// TIA Portal V20 export
ORGANIZATION_BLOCK "Startup"   // OB100, LAD, Startup
TITLE = "Complete Restart"
// stored: AutoNumber false, IsIECCheckEnabled true, SetENOAutomatically true
   VAR_INPUT
      LostRetentive : Bool;   // True if retentive data are lost
      LostRTC : Bool;   // True if date and time are lost
   END_VAR
   VAR_TEMP
      tempError : Bool;
      tempStatus : Word;
      tempDiagnostics : "LAF_typeDiagnosticsSimple";
   END_VAR
BEGIN

REGION Network 1: Set first cycle bit
   // Set the first cycle signal
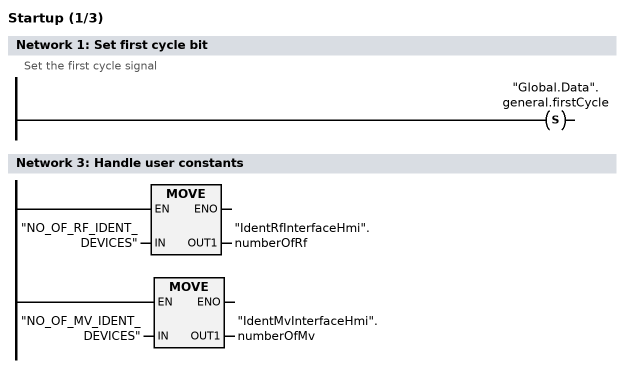
   RUNG wire#powerrail
      S_Coil( "Global.Data".general.firstCycle )
   END_RUNG
   // the same network as SCL:
   "Global.Data".general.firstCycle := TRUE;
END_REGION

REGION Network 2: Enable global power
   // Set global power to true by default. This can be adjusted depending on the user requirement for a specific machine.
END_REGION

REGION Network 3: Handle user constants
   RUNG wire#powerrail
      Move(in := "NO_OF_RF_IDENT_DEVICES", out1 => "IdentRfInterfaceHmi".numberOfRf)
   END_RUNG
   RUNG wire#powerrail
      Move(in := "NO_OF_MV_IDENT_DEVICES", out1 => "IdentMvInterfaceHmi".numberOfMv)
   END_RUNG
   // the same network as SCL:
   "IdentRfInterfaceHmi".numberOfRf := "NO_OF_RF_IDENT_DEVICES";
   "IdentMvInterfaceHmi".numberOfMv := "NO_OF_MV_IDENT_DEVICES";
END_REGION

REGION Network 4: Set drive objects for drive diagnostic
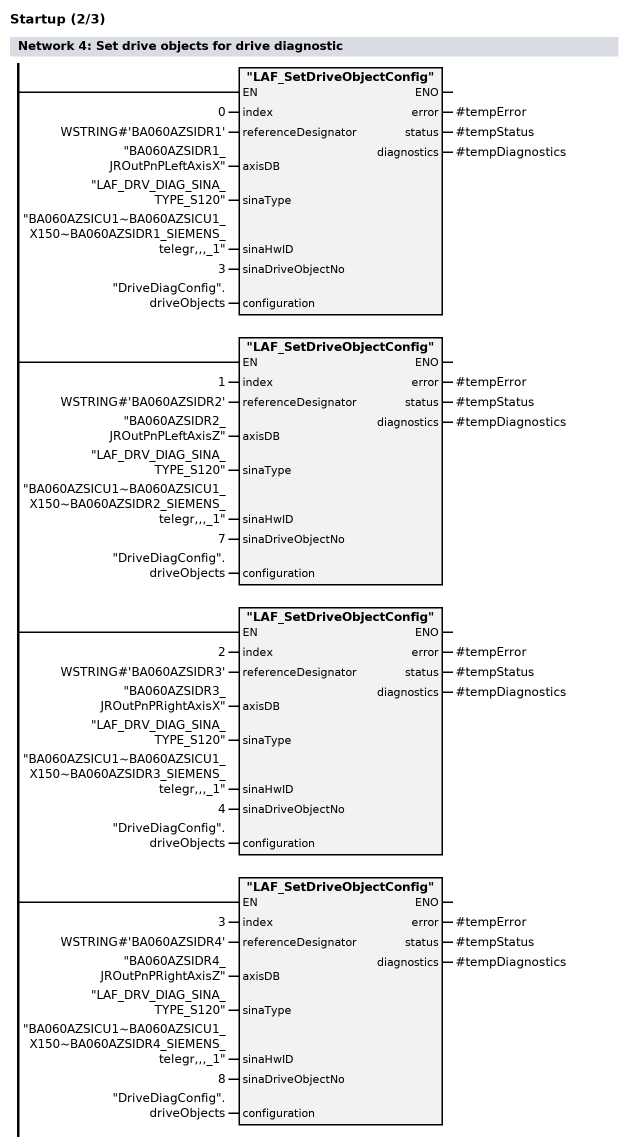
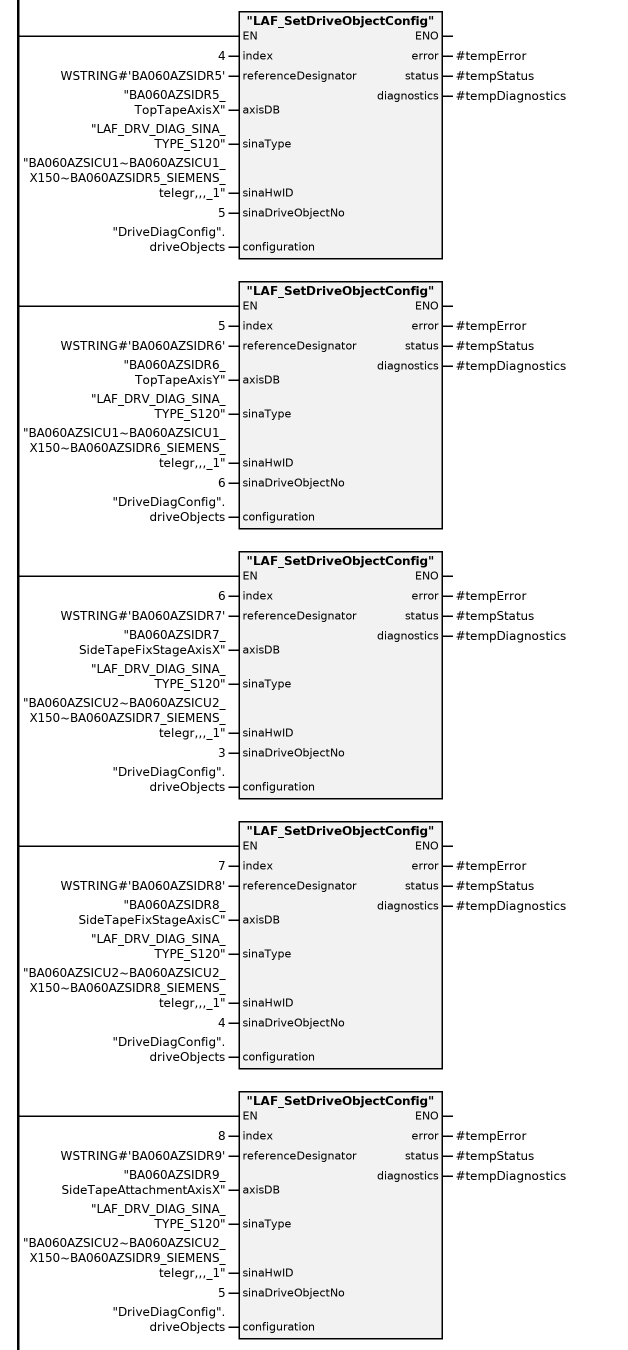
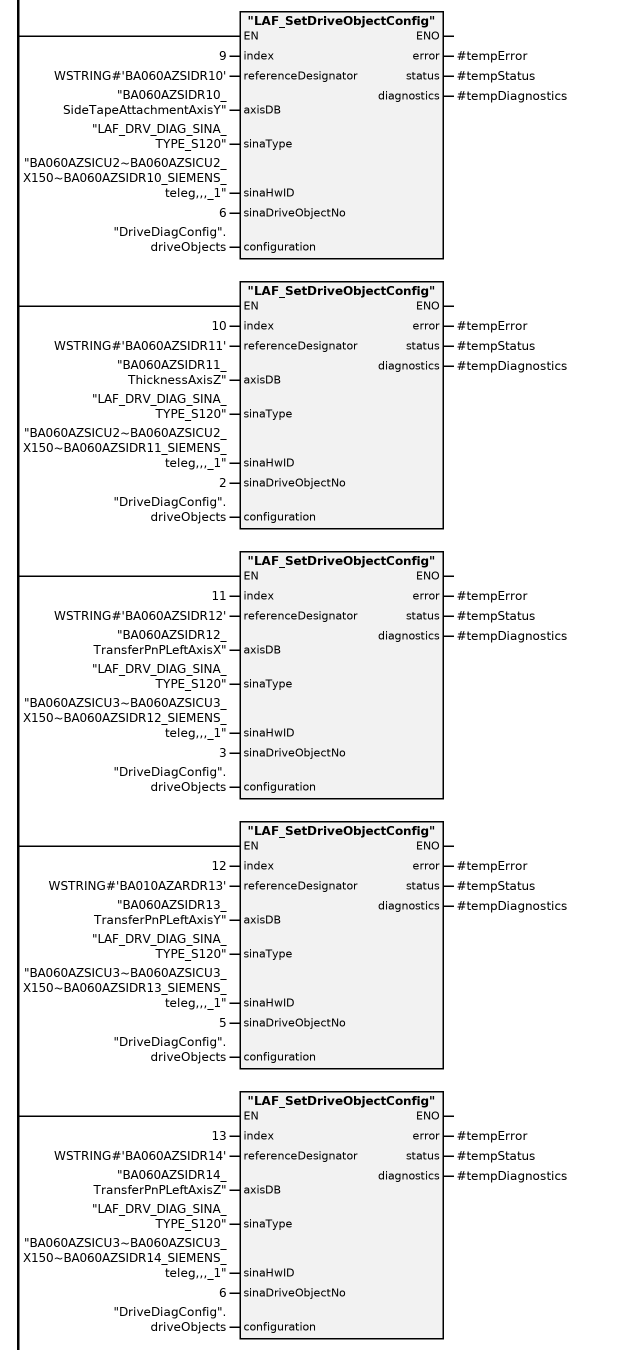
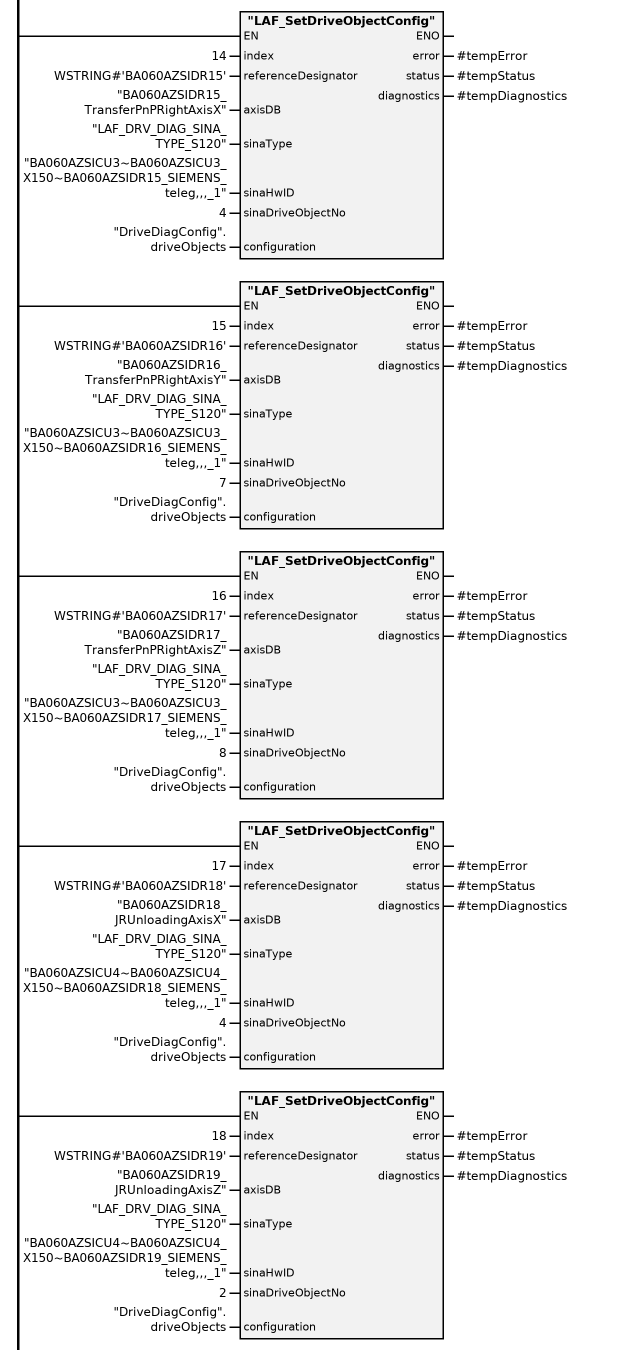
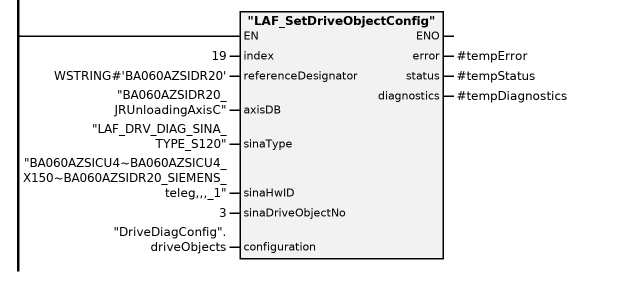
   RUNG wire#powerrail
      "LAF_SetDriveObjectConfig"(index := 0, referenceDesignator := WSTRING#'BA060AZSIDR1', axisDB := "BA060AZSIDR1_JROutPnPLeftAxisX", sinaType := "LAF_DRV_DIAG_SINA_TYPE_S120", sinaHwID := "BA060AZSICU1~BA060AZSICU1_X150~BA060AZSIDR1_SIEMENS_telegr,,,_1", sinaDriveObjectNo := 3, configuration := "DriveDiagConfig".driveObjects, error => #tempError, status => #tempStatus, diagnostics => #tempDiagnostics)
   END_RUNG
   RUNG wire#powerrail
      "LAF_SetDriveObjectConfig"(index := 1, referenceDesignator := WSTRING#'BA060AZSIDR2', axisDB := "BA060AZSIDR2_JROutPnPLeftAxisZ", sinaType := "LAF_DRV_DIAG_SINA_TYPE_S120", sinaHwID := "BA060AZSICU1~BA060AZSICU1_X150~BA060AZSIDR2_SIEMENS_telegr,,,_1", sinaDriveObjectNo := 7, configuration := "DriveDiagConfig".driveObjects, error => #tempError, status => #tempStatus, diagnostics => #tempDiagnostics)
   END_RUNG
   RUNG wire#powerrail
      "LAF_SetDriveObjectConfig"(index := 2, referenceDesignator := WSTRING#'BA060AZSIDR3', axisDB := "BA060AZSIDR3_JROutPnPRightAxisX", sinaType := "LAF_DRV_DIAG_SINA_TYPE_S120", sinaHwID := "BA060AZSICU1~BA060AZSICU1_X150~BA060AZSIDR3_SIEMENS_telegr,,,_1", sinaDriveObjectNo := 4, configuration := "DriveDiagConfig".driveObjects, error => #tempError, status => #tempStatus, diagnostics => #tempDiagnostics)
   END_RUNG
   RUNG wire#powerrail
      "LAF_SetDriveObjectConfig"(index := 3, referenceDesignator := WSTRING#'BA060AZSIDR4', axisDB := "BA060AZSIDR4_JROutPnPRightAxisZ", sinaType := "LAF_DRV_DIAG_SINA_TYPE_S120", sinaHwID := "BA060AZSICU1~BA060AZSICU1_X150~BA060AZSIDR4_SIEMENS_telegr,,,_1", sinaDriveObjectNo := 8, configuration := "DriveDiagConfig".driveObjects, error => #tempError, status => #tempStatus, diagnostics => #tempDiagnostics)
   END_RUNG
   RUNG wire#powerrail
      "LAF_SetDriveObjectConfig"(index := 4, referenceDesignator := WSTRING#'BA060AZSIDR5', axisDB := "BA060AZSIDR5_TopTapeAxisX", sinaType := "LAF_DRV_DIAG_SINA_TYPE_S120", sinaHwID := "BA060AZSICU1~BA060AZSICU1_X150~BA060AZSIDR5_SIEMENS_telegr,,,_1", sinaDriveObjectNo := 5, configuration := "DriveDiagConfig".driveObjects, error => #tempError, status => #tempStatus, diagnostics => #tempDiagnostics)
   END_RUNG
   RUNG wire#powerrail
      "LAF_SetDriveObjectConfig"(index := 5, referenceDesignator := WSTRING#'BA060AZSIDR6', axisDB := "BA060AZSIDR6_TopTapeAxisY", sinaType := "LAF_DRV_DIAG_SINA_TYPE_S120", sinaHwID := "BA060AZSICU1~BA060AZSICU1_X150~BA060AZSIDR6_SIEMENS_telegr,,,_1", sinaDriveObjectNo := 6, configuration := "DriveDiagConfig".driveObjects, error => #tempError, status => #tempStatus, diagnostics => #tempDiagnostics)
   END_RUNG
   RUNG wire#powerrail
      "LAF_SetDriveObjectConfig"(index := 6, referenceDesignator := WSTRING#'BA060AZSIDR7', axisDB := "BA060AZSIDR7_SideTapeFixStageAxisX", sinaType := "LAF_DRV_DIAG_SINA_TYPE_S120", sinaHwID := "BA060AZSICU2~BA060AZSICU2_X150~BA060AZSIDR7_SIEMENS_telegr,,,_1", sinaDriveObjectNo := 3, configuration := "DriveDiagConfig".driveObjects, error => #tempError, status => #tempStatus, diagnostics => #tempDiagnostics)
   END_RUNG
   RUNG wire#powerrail
      "LAF_SetDriveObjectConfig"(index := 7, referenceDesignator := WSTRING#'BA060AZSIDR8', axisDB := "BA060AZSIDR8_SideTapeFixStageAxisC", sinaType := "LAF_DRV_DIAG_SINA_TYPE_S120", sinaHwID := "BA060AZSICU2~BA060AZSICU2_X150~BA060AZSIDR8_SIEMENS_telegr,,,_1", sinaDriveObjectNo := 4, configuration := "DriveDiagConfig".driveObjects, error => #tempError, status => #tempStatus, diagnostics => #tempDiagnostics)
   END_RUNG
   RUNG wire#powerrail
      "LAF_SetDriveObjectConfig"(index := 8, referenceDesignator := WSTRING#'BA060AZSIDR9', axisDB := "BA060AZSIDR9_SideTapeAttachmentAxisX", sinaType := "LAF_DRV_DIAG_SINA_TYPE_S120", sinaHwID := "BA060AZSICU2~BA060AZSICU2_X150~BA060AZSIDR9_SIEMENS_telegr,,,_1", sinaDriveObjectNo := 5, configuration := "DriveDiagConfig".driveObjects, error => #tempError, status => #tempStatus, diagnostics => #tempDiagnostics)
   END_RUNG
   RUNG wire#powerrail
      "LAF_SetDriveObjectConfig"(index := 9, referenceDesignator := WSTRING#'BA060AZSIDR10', axisDB := "BA060AZSIDR10_SideTapeAttachmentAxisY", sinaType := "LAF_DRV_DIAG_SINA_TYPE_S120", sinaHwID := "BA060AZSICU2~BA060AZSICU2_X150~BA060AZSIDR10_SIEMENS_teleg,,,_1", sinaDriveObjectNo := 6, configuration := "DriveDiagConfig".driveObjects, error => #tempError, status => #tempStatus, diagnostics => #tempDiagnostics)
   END_RUNG
   RUNG wire#powerrail
      "LAF_SetDriveObjectConfig"(index := 10, referenceDesignator := WSTRING#'BA060AZSIDR11', axisDB := "BA060AZSIDR11_ThicknessAxisZ", sinaType := "LAF_DRV_DIAG_SINA_TYPE_S120", sinaHwID := "BA060AZSICU2~BA060AZSICU2_X150~BA060AZSIDR11_SIEMENS_teleg,,,_1", sinaDriveObjectNo := 2, configuration := "DriveDiagConfig".driveObjects, error => #tempError, status => #tempStatus, diagnostics => #tempDiagnostics)
   END_RUNG
   RUNG wire#powerrail
      "LAF_SetDriveObjectConfig"(index := 11, referenceDesignator := WSTRING#'BA060AZSIDR12', axisDB := "BA060AZSIDR12_TransferPnPLeftAxisX", sinaType := "LAF_DRV_DIAG_SINA_TYPE_S120", sinaHwID := "BA060AZSICU3~BA060AZSICU3_X150~BA060AZSIDR12_SIEMENS_teleg,,,_1", sinaDriveObjectNo := 3, configuration := "DriveDiagConfig".driveObjects, error => #tempError, status => #tempStatus, diagnostics => #tempDiagnostics)
   END_RUNG
   RUNG wire#powerrail
      "LAF_SetDriveObjectConfig"(index := 12, referenceDesignator := WSTRING#'BA010AZARDR13', axisDB := "BA060AZSIDR13_TransferPnPLeftAxisY", sinaType := "LAF_DRV_DIAG_SINA_TYPE_S120", sinaHwID := "BA060AZSICU3~BA060AZSICU3_X150~BA060AZSIDR13_SIEMENS_teleg,,,_1", sinaDriveObjectNo := 5, configuration := "DriveDiagConfig".driveObjects, error => #tempError, status => #tempStatus, diagnostics => #tempDiagnostics)
   END_RUNG
   RUNG wire#powerrail
      "LAF_SetDriveObjectConfig"(index := 13, referenceDesignator := WSTRING#'BA060AZSIDR14', axisDB := "BA060AZSIDR14_TransferPnPLeftAxisZ", sinaType := "LAF_DRV_DIAG_SINA_TYPE_S120", sinaHwID := "BA060AZSICU3~BA060AZSICU3_X150~BA060AZSIDR14_SIEMENS_teleg,,,_1", sinaDriveObjectNo := 6, configuration := "DriveDiagConfig".driveObjects, error => #tempError, status => #tempStatus, diagnostics => #tempDiagnostics)
   END_RUNG
   RUNG wire#powerrail
      "LAF_SetDriveObjectConfig"(index := 14, referenceDesignator := WSTRING#'BA060AZSIDR15', axisDB := "BA060AZSIDR15_TransferPnPRightAxisX", sinaType := "LAF_DRV_DIAG_SINA_TYPE_S120", sinaHwID := "BA060AZSICU3~BA060AZSICU3_X150~BA060AZSIDR15_SIEMENS_teleg,,,_1", sinaDriveObjectNo := 4, configuration := "DriveDiagConfig".driveObjects, error => #tempError, status => #tempStatus, diagnostics => #tempDiagnostics)
   END_RUNG
   RUNG wire#powerrail
      "LAF_SetDriveObjectConfig"(index := 15, referenceDesignator := WSTRING#'BA060AZSIDR16', axisDB := "BA060AZSIDR16_TransferPnPRightAxisY", sinaType := "LAF_DRV_DIAG_SINA_TYPE_S120", sinaHwID := "BA060AZSICU3~BA060AZSICU3_X150~BA060AZSIDR16_SIEMENS_teleg,,,_1", sinaDriveObjectNo := 7, configuration := "DriveDiagConfig".driveObjects, error => #tempError, status => #tempStatus, diagnostics => #tempDiagnostics)
   END_RUNG
   RUNG wire#powerrail
      "LAF_SetDriveObjectConfig"(index := 16, referenceDesignator := WSTRING#'BA060AZSIDR17', axisDB := "BA060AZSIDR17_TransferPnPRightAxisZ", sinaType := "LAF_DRV_DIAG_SINA_TYPE_S120", sinaHwID := "BA060AZSICU3~BA060AZSICU3_X150~BA060AZSIDR17_SIEMENS_teleg,,,_1", sinaDriveObjectNo := 8, configuration := "DriveDiagConfig".driveObjects, error => #tempError, status => #tempStatus, diagnostics => #tempDiagnostics)
   END_RUNG
   RUNG wire#powerrail
      "LAF_SetDriveObjectConfig"(index := 17, referenceDesignator := WSTRING#'BA060AZSIDR18', axisDB := "BA060AZSIDR18_JRUnloadingAxisX", sinaType := "LAF_DRV_DIAG_SINA_TYPE_S120", sinaHwID := "BA060AZSICU4~BA060AZSICU4_X150~BA060AZSIDR18_SIEMENS_teleg,,,_1", sinaDriveObjectNo := 4, configuration := "DriveDiagConfig".driveObjects, error => #tempError, status => #tempStatus, diagnostics => #tempDiagnostics)
   END_RUNG
   RUNG wire#powerrail
      "LAF_SetDriveObjectConfig"(index := 18, referenceDesignator := WSTRING#'BA060AZSIDR19', axisDB := "BA060AZSIDR19_JRUnloadingAxisZ", sinaType := "LAF_DRV_DIAG_SINA_TYPE_S120", sinaHwID := "BA060AZSICU4~BA060AZSICU4_X150~BA060AZSIDR19_SIEMENS_teleg,,,_1", sinaDriveObjectNo := 2, configuration := "DriveDiagConfig".driveObjects, error => #tempError, status => #tempStatus, diagnostics => #tempDiagnostics)
   END_RUNG
   RUNG wire#powerrail
      "LAF_SetDriveObjectConfig"(index := 19, referenceDesignator := WSTRING#'BA060AZSIDR20', axisDB := "BA060AZSIDR20_JRUnloadingAxisC", sinaType := "LAF_DRV_DIAG_SINA_TYPE_S120", sinaHwID := "BA060AZSICU4~BA060AZSICU4_X150~BA060AZSIDR20_SIEMENS_teleg,,,_1", sinaDriveObjectNo := 3, configuration := "DriveDiagConfig".driveObjects, error => #tempError, status => #tempStatus, diagnostics => #tempDiagnostics)
   END_RUNG
   // the same network as SCL:
   "LAF_SetDriveObjectConfig"(index := 0,
                           referenceDesignator := WSTRING#'BA060AZSIDR1',
                           axisDB := "BA060AZSIDR1_JROutPnPLeftAxisX",
                           sinaType := "LAF_DRV_DIAG_SINA_TYPE_S120",
                           sinaHwID := "BA060AZSICU1~BA060AZSICU1_X150~BA060AZSIDR1_SIEMENS_telegr,,,_1",
                           sinaDriveObjectNo := 3,
                           configuration := "DriveDiagConfig".driveObjects,
                           error => #tempError,
                           status => #tempStatus,
                           diagnostics => #tempDiagnostics);
   "LAF_SetDriveObjectConfig"(index := 1,
                           referenceDesignator := WSTRING#'BA060AZSIDR2',
                           axisDB := "BA060AZSIDR2_JROutPnPLeftAxisZ",
                           sinaType := "LAF_DRV_DIAG_SINA_TYPE_S120",
                           sinaHwID := "BA060AZSICU1~BA060AZSICU1_X150~BA060AZSIDR2_SIEMENS_telegr,,,_1",
                           sinaDriveObjectNo := 7,
                           configuration := "DriveDiagConfig".driveObjects,
                           error => #tempError,
                           status => #tempStatus,
                           diagnostics => #tempDiagnostics);
   "LAF_SetDriveObjectConfig"(index := 2,
                           referenceDesignator := WSTRING#'BA060AZSIDR3',
                           axisDB := "BA060AZSIDR3_JROutPnPRightAxisX",
                           sinaType := "LAF_DRV_DIAG_SINA_TYPE_S120",
                           sinaHwID := "BA060AZSICU1~BA060AZSICU1_X150~BA060AZSIDR3_SIEMENS_telegr,,,_1",
                           sinaDriveObjectNo := 4,
                           configuration := "DriveDiagConfig".driveObjects,
                           error => #tempError,
                           status => #tempStatus,
                           diagnostics => #tempDiagnostics);
   "LAF_SetDriveObjectConfig"(index := 3,
                           referenceDesignator := WSTRING#'BA060AZSIDR4',
                           axisDB := "BA060AZSIDR4_JROutPnPRightAxisZ",
                           sinaType := "LAF_DRV_DIAG_SINA_TYPE_S120",
                           sinaHwID := "BA060AZSICU1~BA060AZSICU1_X150~BA060AZSIDR4_SIEMENS_telegr,,,_1",
                           sinaDriveObjectNo := 8,
                           configuration := "DriveDiagConfig".driveObjects,
                           error => #tempError,
                           status => #tempStatus,
                           diagnostics => #tempDiagnostics);
   "LAF_SetDriveObjectConfig"(index := 4,
                           referenceDesignator := WSTRING#'BA060AZSIDR5',
                           axisDB := "BA060AZSIDR5_TopTapeAxisX",
                           sinaType := "LAF_DRV_DIAG_SINA_TYPE_S120",
                           sinaHwID := "BA060AZSICU1~BA060AZSICU1_X150~BA060AZSIDR5_SIEMENS_telegr,,,_1",
                           sinaDriveObjectNo := 5,
                           configuration := "DriveDiagConfig".driveObjects,
                           error => #tempError,
                           status => #tempStatus,
                           diagnostics => #tempDiagnostics);
   "LAF_SetDriveObjectConfig"(index := 5,
                           referenceDesignator := WSTRING#'BA060AZSIDR6',
                           axisDB := "BA060AZSIDR6_TopTapeAxisY",
                           sinaType := "LAF_DRV_DIAG_SINA_TYPE_S120",
                           sinaHwID := "BA060AZSICU1~BA060AZSICU1_X150~BA060AZSIDR6_SIEMENS_telegr,,,_1",
                           sinaDriveObjectNo := 6,
                           configuration := "DriveDiagConfig".driveObjects,
                           error => #tempError,
                           status => #tempStatus,
                           diagnostics => #tempDiagnostics);
   "LAF_SetDriveObjectConfig"(index := 6,
                           referenceDesignator := WSTRING#'BA060AZSIDR7',
                           axisDB := "BA060AZSIDR7_SideTapeFixStageAxisX",
                           sinaType := "LAF_DRV_DIAG_SINA_TYPE_S120",
                           sinaHwID := "BA060AZSICU2~BA060AZSICU2_X150~BA060AZSIDR7_SIEMENS_telegr,,,_1",
                           sinaDriveObjectNo := 3,
                           configuration := "DriveDiagConfig".driveObjects,
                           error => #tempError,
                           status => #tempStatus,
                           diagnostics => #tempDiagnostics);
   "LAF_SetDriveObjectConfig"(index := 7,
                           referenceDesignator := WSTRING#'BA060AZSIDR8',
                           axisDB := "BA060AZSIDR8_SideTapeFixStageAxisC",
                           sinaType := "LAF_DRV_DIAG_SINA_TYPE_S120",
                           sinaHwID := "BA060AZSICU2~BA060AZSICU2_X150~BA060AZSIDR8_SIEMENS_telegr,,,_1",
                           sinaDriveObjectNo := 4,
                           configuration := "DriveDiagConfig".driveObjects,
                           error => #tempError,
                           status => #tempStatus,
                           diagnostics => #tempDiagnostics);
   "LAF_SetDriveObjectConfig"(index := 8,
                           referenceDesignator := WSTRING#'BA060AZSIDR9',
                           axisDB := "BA060AZSIDR9_SideTapeAttachmentAxisX",
                           sinaType := "LAF_DRV_DIAG_SINA_TYPE_S120",
                           sinaHwID := "BA060AZSICU2~BA060AZSICU2_X150~BA060AZSIDR9_SIEMENS_telegr,,,_1",
                           sinaDriveObjectNo := 5,
                           configuration := "DriveDiagConfig".driveObjects,
                           error => #tempError,
                           status => #tempStatus,
                           diagnostics => #tempDiagnostics);
   "LAF_SetDriveObjectConfig"(index := 9,
                           referenceDesignator := WSTRING#'BA060AZSIDR10',
                           axisDB := "BA060AZSIDR10_SideTapeAttachmentAxisY",
                           sinaType := "LAF_DRV_DIAG_SINA_TYPE_S120",
                           sinaHwID := "BA060AZSICU2~BA060AZSICU2_X150~BA060AZSIDR10_SIEMENS_teleg,,,_1",
                           sinaDriveObjectNo := 6,
                           configuration := "DriveDiagConfig".driveObjects,
                           error => #tempError,
                           status => #tempStatus,
                           diagnostics => #tempDiagnostics);
   "LAF_SetDriveObjectConfig"(index := 10,
                           referenceDesignator := WSTRING#'BA060AZSIDR11',
                           axisDB := "BA060AZSIDR11_ThicknessAxisZ",
                           sinaType := "LAF_DRV_DIAG_SINA_TYPE_S120",
                           sinaHwID := "BA060AZSICU2~BA060AZSICU2_X150~BA060AZSIDR11_SIEMENS_teleg,,,_1",
                           sinaDriveObjectNo := 2,
                           configuration := "DriveDiagConfig".driveObjects,
                           error => #tempError,
                           status => #tempStatus,
                           diagnostics => #tempDiagnostics);
   "LAF_SetDriveObjectConfig"(index := 11,
                           referenceDesignator := WSTRING#'BA060AZSIDR12',
                           axisDB := "BA060AZSIDR12_TransferPnPLeftAxisX",
                           sinaType := "LAF_DRV_DIAG_SINA_TYPE_S120",
                           sinaHwID := "BA060AZSICU3~BA060AZSICU3_X150~BA060AZSIDR12_SIEMENS_teleg,,,_1",
                           sinaDriveObjectNo := 3,
                           configuration := "DriveDiagConfig".driveObjects,
                           error => #tempError,
                           status => #tempStatus,
                           diagnostics => #tempDiagnostics);
   "LAF_SetDriveObjectConfig"(index := 12,
                           referenceDesignator := WSTRING#'BA010AZARDR13',
                           axisDB := "BA060AZSIDR13_TransferPnPLeftAxisY",
                           sinaType := "LAF_DRV_DIAG_SINA_TYPE_S120",
                           sinaHwID := "BA060AZSICU3~BA060AZSICU3_X150~BA060AZSIDR13_SIEMENS_teleg,,,_1",
                           sinaDriveObjectNo := 5,
                           configuration := "DriveDiagConfig".driveObjects,
                           error => #tempError,
                           status => #tempStatus,
                           diagnostics => #tempDiagnostics);
   "LAF_SetDriveObjectConfig"(index := 13,
                           referenceDesignator := WSTRING#'BA060AZSIDR14',
                           axisDB := "BA060AZSIDR14_TransferPnPLeftAxisZ",
                           sinaType := "LAF_DRV_DIAG_SINA_TYPE_S120",
                           sinaHwID := "BA060AZSICU3~BA060AZSICU3_X150~BA060AZSIDR14_SIEMENS_teleg,,,_1",
                           sinaDriveObjectNo := 6,
                           configuration := "DriveDiagConfig".driveObjects,
                           error => #tempError,
                           status => #tempStatus,
                           diagnostics => #tempDiagnostics);
   "LAF_SetDriveObjectConfig"(index := 14,
                           referenceDesignator := WSTRING#'BA060AZSIDR15',
                           axisDB := "BA060AZSIDR15_TransferPnPRightAxisX",
                           sinaType := "LAF_DRV_DIAG_SINA_TYPE_S120",
                           sinaHwID := "BA060AZSICU3~BA060AZSICU3_X150~BA060AZSIDR15_SIEMENS_teleg,,,_1",
                           sinaDriveObjectNo := 4,
                           configuration := "DriveDiagConfig".driveObjects,
                           error => #tempError,
                           status => #tempStatus,
                           diagnostics => #tempDiagnostics);
   "LAF_SetDriveObjectConfig"(index := 15,
                           referenceDesignator := WSTRING#'BA060AZSIDR16',
                           axisDB := "BA060AZSIDR16_TransferPnPRightAxisY",
                           sinaType := "LAF_DRV_DIAG_SINA_TYPE_S120",
                           sinaHwID := "BA060AZSICU3~BA060AZSICU3_X150~BA060AZSIDR16_SIEMENS_teleg,,,_1",
                           sinaDriveObjectNo := 7,
                           configuration := "DriveDiagConfig".driveObjects,
                           error => #tempError,
                           status => #tempStatus,
                           diagnostics => #tempDiagnostics);
   "LAF_SetDriveObjectConfig"(index := 16,
                           referenceDesignator := WSTRING#'BA060AZSIDR17',
                           axisDB := "BA060AZSIDR17_TransferPnPRightAxisZ",
                           sinaType := "LAF_DRV_DIAG_SINA_TYPE_S120",
                           sinaHwID := "BA060AZSICU3~BA060AZSICU3_X150~BA060AZSIDR17_SIEMENS_teleg,,,_1",
                           sinaDriveObjectNo := 8,
                           configuration := "DriveDiagConfig".driveObjects,
                           error => #tempError,
                           status => #tempStatus,
                           diagnostics => #tempDiagnostics);
   "LAF_SetDriveObjectConfig"(index := 17,
                           referenceDesignator := WSTRING#'BA060AZSIDR18',
                           axisDB := "BA060AZSIDR18_JRUnloadingAxisX",
                           sinaType := "LAF_DRV_DIAG_SINA_TYPE_S120",
                           sinaHwID := "BA060AZSICU4~BA060AZSICU4_X150~BA060AZSIDR18_SIEMENS_teleg,,,_1",
                           sinaDriveObjectNo := 4,
                           configuration := "DriveDiagConfig".driveObjects,
                           error => #tempError,
                           status => #tempStatus,
                           diagnostics => #tempDiagnostics);
   "LAF_SetDriveObjectConfig"(index := 18,
                           referenceDesignator := WSTRING#'BA060AZSIDR19',
                           axisDB := "BA060AZSIDR19_JRUnloadingAxisZ",
                           sinaType := "LAF_DRV_DIAG_SINA_TYPE_S120",
                           sinaHwID := "BA060AZSICU4~BA060AZSICU4_X150~BA060AZSIDR19_SIEMENS_teleg,,,_1",
                           sinaDriveObjectNo := 2,
                           configuration := "DriveDiagConfig".driveObjects,
                           error => #tempError,
                           status => #tempStatus,
                           diagnostics => #tempDiagnostics);
   "LAF_SetDriveObjectConfig"(index := 19,
                           referenceDesignator := WSTRING#'BA060AZSIDR20',
                           axisDB := "BA060AZSIDR20_JRUnloadingAxisC",
                           sinaType := "LAF_DRV_DIAG_SINA_TYPE_S120",
                           sinaHwID := "BA060AZSICU4~BA060AZSICU4_X150~BA060AZSIDR20_SIEMENS_teleg,,,_1",
                           sinaDriveObjectNo := 3,
                           configuration := "DriveDiagConfig".driveObjects,
                           error => #tempError,
                           status => #tempStatus,
                           diagnostics => #tempDiagnostics);
END_REGION

REGION Network 5: Manual Operation Line
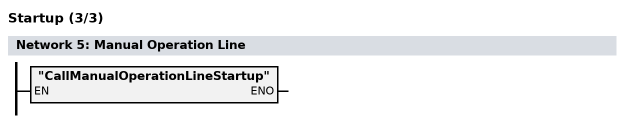
   RUNG wire#powerrail
      "CallManualOperationLineStartup"()
   END_RUNG
   // the same network as SCL:
   "CallManualOperationLineStartup"();
END_REGION

REGION Network 6 (SCL): Configuration Set Position
   //DR01
   "Unit1.Em2.HmiInterface".cmJROutPnPLeftAxisX.configuration.setPositions := "AxisDataBackUp_DB".DR1."configuration.setPositions";
   //Unit1.Em2.HmiInterface.cm.softcam.jrOutPnPLeftAxisX := "AxisDataBackUp_DB".DR1.softcam;


   //DR02
   "Unit1.Em2.HmiInterface".cmJROutPnPLeftAxisZ.configuration.setPositions := "AxisDataBackUp_DB".DR2."configuration.setPositions";
   //Unit1.Em2.HmiInterface.cm.softcam.jrOutPnPLeftAxisZ := "AxisDataBackUp_DB".DR2.softcam;


   //DR03
   "Unit1.Em2.HmiInterface".cmJROutPnPRightAxisX.configuration.setPositions := "AxisDataBackUp_DB".DR3."configuration.setPositions";
   //Unit1.Em2.HmiInterface.cm.softcam.jrOutPnPRightAxisX := "AxisDataBackUp_DB".DR3.softcam;


   //DR04
   "Unit1.Em2.HmiInterface".cmJROutPnPRightAxisZ.configuration.setPositions := "AxisDataBackUp_DB".DR4."configuration.setPositions";
   //Unit1.Em2.HmiInterface.cm.softcam.jrOutPnPRightAxisZ := "AxisDataBackUp_DB".DR4.softcam;


   //DR05
   "Unit1.Em3.HmiInterface".cmTopTapeAxisX.configuration.setPositions := "AxisDataBackUp_DB".DR5."configuration.setPositions";
   //Unit1.Em3.HmiInterface.cm.softcam.topTapeAxisX := "AxisDataBackUp_DB".DR5.softcam;


   //DR06
   "Unit1.Em3.HmiInterface".cmTopTapeAxisY.configuration.setPositions := "AxisDataBackUp_DB".DR6."configuration.setPositions";
   //Unit1.Em3.HmiInterface.cm.softcam.topTapeAxisY := "AxisDataBackUp_DB".DR6.softcam;


   //DR07
   "Unit1.Em4.HmiInterface".cmSideTapeFixStageAxisX.configuration.setPositions := "AxisDataBackUp_DB".DR7."configuration.setPositions";
   //Unit1.Em4.HmiInterface.cm.softcam.sideTapeFixStageAxisX := "AxisDataBackUp_DB".DR7.softcam;


   //DR08
   "Unit1.Em4.HmiInterface".cmSideTapeFixStageAxisC.configuration.setPositions := "AxisDataBackUp_DB".DR8."configuration.setPositions";
   //Unit1.Em4.HmiInterface.cm.softcam.sideTapeFixStageAxisC := "AxisDataBackUp_DB".DR8.softcam;


   //DR09
   "Unit1.Em4.HmiInterface".cmSideTapeAttachmentAxisX.configuration.setPositions := "AxisDataBackUp_DB".DR9."configuration.setPositions";
   //Unit1.Em4.HmiInterface.cm.softcam.sideTapeAttachmentAxisX := "AxisDataBackUp_DB".DR9.softcam;


   //DR10
   "Unit1.Em4.HmiInterface".cmSideTapeAttachmentAxisY.configuration.setPositions := "AxisDataBackUp_DB".DR10."configuration.setPositions";
   //Unit1.Em4.HmiInterface.cm.softcam.sideTapeAttachmentAxisY := "AxisDataBackUp_DB".DR10.softcam;


   //DR11
   "Unit1.Em8.HmiInterface".cmThicknessAxisZ.configuration.setPositions := "AxisDataBackUp_DB".DR11."configuration.setPositions";
   //Unit1.Em8.HmiInterface.cm.softcam.thicknessAxisZ := "AxisDataBackUp_DB".DR11.softcam;


   //DR12
   "Unit1.Em5.HmiInterface".cmTransferPnPLeftAxisX.configuration.setPositions := "AxisDataBackUp_DB".DR12."configuration.setPositions";
   //Unit1.Em5.HmiInterface.cm.softcam.transferPnPLeftAxisX := "AxisDataBackUp_DB".DR12.softcam;

   //DR13
   "Unit1.Em5.HmiInterface".cmTransferPnPLeftAxisY.configuration.setPositions := "AxisDataBackUp_DB".DR13."configuration.setPositions";
   //Unit1.Em5.HmiInterface.cm.softcam.transferPnPLeftAxisY := "AxisDataBackUp_DB".DR13.softcam;


   //DR14
   "Unit1.Em5.HmiInterface".cmTransferPnPLeftAxisZ.configuration.setPositions := "AxisDataBackUp_DB".DR14."configuration.setPositions";
   //Unit1.Em5.HmiInterface.cm.softcam.transferPnPLeftAxisZ := "AxisDataBackUp_DB".DR14.softcam;


   //DR15
   "Unit1.Em5.HmiInterface".cmTransferPnPRightAxisX.configuration.setPositions := "AxisDataBackUp_DB".DR15."configuration.setPositions";
   //Unit1.Em5.HmiInterface.cm.softcam.transferPnPRightAxisX := "AxisDataBackUp_DB".DR15.softcam;


   //DR16
   "Unit1.Em5.HmiInterface".cmTransferPnPRightAxisY.configuration.setPositions := "AxisDataBackUp_DB".DR16."configuration.setPositions";
   //Unit1.Em5.HmiInterface.cm.softcam.transferPnPRightAxisY := "AxisDataBackUp_DB".DR16.softcam;


   //DR17
   "Unit1.Em5.HmiInterface".cmTransferPnPRightAxisZ.configuration.setPositions := "AxisDataBackUp_DB".DR17."configuration.setPositions";
   //Unit1.Em5.HmiInterface.cm.softcam.transferPnPRightAxisZ := "AxisDataBackUp_DB".DR17.softcam;


   //DR18
   "Unit1.Em13.HmiInterface".cmJRUnloadingPnPAxisX.configuration.setPositions := "AxisDataBackUp_DB".DR18."configuration.setPositions";
   //Unit1.Em13.HmiInterface.cm.softcam.jrUnloadingPnPAxisX := "AxisDataBackUp_DB".DR18.softcam;


   //DR19
   "Unit1.Em13.HmiInterface".cmJRUnloadingPnPAxisZ.configuration.setPositions := "AxisDataBackUp_DB".DR19."configuration.setPositions";
   //Unit1.Em13.HmiInterface.cm.softcam.jrUnloadingPnPAxisZ := "AxisDataBackUp_DB".DR19.softcam;


   //DR20
   "Unit1.Em13.HmiInterface".cmJRUnloadingPnPAxisC.configuration.setPositions := "AxisDataBackUp_DB".DR20."configuration.setPositions";
   //Unit1.Em13.HmiInterface.cm.softcam.jrUnloadingPnPAxisC := "AxisDataBackUp_DB".DR20.softcam;
END_REGION
END_ORGANIZATION_BLOCK
